Staubli VAL3: page.pgx

public program page(string& menuname[], num index)
// set all the page
begin
  //
  //  PAGE
  //
  //,,,,,,,,,,,,,,,,,,,,,,,
  //  go home setting
  //,,,,,,,,,,,,,,,,,,,,,,,
  //
  //  HOME PAGE
  //
  //
  if index>=300 and index<=301
    title("< 一键回零设置界面 > "+menuname)
  endIf

  //,,,,,,,,,,,,,,,,,,,,
  //  CYCLE
  //,,,,,,,,,,,,,,,,,,,,
  //  if index>=20 and index<=29
  //    title("< Production Page >")
  //  endIf
  //  if index>=200 and index<=209
  //    title("< Simulation >")
  //  endIf
  //  if index>=210 and index<=219
  //    title ("< Stepping Simulation >")
  //  endIf
  //
  //  MENU
  //
  menuname=""
  //,,,,,,,,,,,,,,,,,,,,
  //  KERNEL
  //,,,,,,,,,,,,,,,,,,,,
  switch index

    case 300
      //
      menuname="测试,,,,,类型,删除,新建"
    break
    case 301
      // cycle
      menuname=",,,,,类型,删除,新建"
    break
    case 302
      // Programmer
      menuname="标记,全选,反选,,,,<<,>>"
    break
    case 303
      // Programmer
      menuname="记录,插入,删除,,,,<<,>>"
    break
    case 304
      // Programmer
      menuname="记录,插入,删除,切换移动方式,,,<<,>>"
    break
  endSwitch
end
